// TwinCAT 3 PLC project LED_Sensors
// ProgramVersion: 3.1.4023.0
// libraries:
//   Tc2_ControllerToolbox, * (Beckhoff Automation GmbH)
//   Tc2_Standard, * (Beckhoff Automation GmbH)
//   Tc2_System, * (Beckhoff Automation GmbH)
//   Tc3_Module, * (Beckhoff Automation GmbH)
// project tree:
//   / PlcTask.TcTTO
//   POUs/ MAIN.TcPOU
// real-time tasks:
//   TASK PlcTask: cycle T#10ms, priority 20, ADS port 350

CONFIGURATION LED_Sensors
    RESOURCE PLC ON TwinCAT3
        TASK PlcTask(INTERVAL := T#10ms, PRIORITY := 20);
        PROGRAM MAIN WITH PlcTask : MAIN;
    END_RESOURCE
END_CONFIGURATION

// ---- POUs/MAIN.TcPOU
PROGRAM MAIN
VAR
	fbPWMSignal : FB_CTRL_PWM_OUT;
	rPWMInput : LREAL;			//[-100,100]
	eMode : E_CTRL_MODE;		//eCTRL_MODE_IDLE:=0,eCTRL_MODE_PASSIVE:=1,eCTRL_MODE_ACTIVE:=2,eCTRL_MODE_RESET:=3,eCTRL_MODE_MANUAL:=4,eCTRL_MODE_TUNE:=5,eCTRL_MODE_SELFTEST:=6,eCTRL_MODE_SYNC_MOVEMENT:=7
	sParameter : ST_CTRL_PWM_OUT_PARAMS;
END_VAR

sParameter.bInstantPWMUpdate := FALSE;
sParameter.tPWMPeriod := T#10S; 				//period of PWM signal
sParameter.tTaskCycleTime := T#10S;				//Task cycle time

fbPWMSignal(
	fPwmInput := rPWMInput,
	eMode := eMode,
	stParams := sParameter,
	bPwmOutBitPos =>,
	bPwmOutBitNeg =>,
	eState =>,
	eErrorId =>,
	bError =>
	);

END_PROGRAM
